FUNCTION_BLOCK ResetXYPos (* Composite Function Block Type *)
  (* Standard: 61499-2 *)
  (* Version 1.0, 2020-02-03, Mario *)
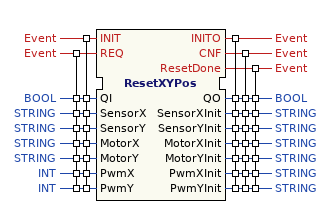
  EVENT_INPUT
    INIT WITH QI, SensorX, SensorY, MotorX, MotorY, PwmX, PwmY; (* Initialization Request *)
    REQ WITH QI, SensorX, SensorY, MotorX, MotorY, PwmX, PwmY; (* Normal Execution Request *)
  END_EVENT
  EVENT_OUTPUT
    INITO WITH QO, SensorXInit, SensorYInit, MotorXInit, MotorYInit, PwmXInit, PwmYInit; (* Initialization Confirm *)
    CNF WITH QO, SensorXInit, SensorYInit, MotorXInit, MotorYInit, PwmXInit, PwmYInit; (* Execution Confirmation *)
    ResetDone WITH QO, SensorXInit, SensorYInit, MotorXInit, MotorYInit, PwmXInit, PwmYInit;
  END_EVENT
  VAR_INPUT
    QI : BOOL; (* Input event qualifier *)
    SensorX : STRING; (* Sensor port to reset X axis *)
    SensorY : STRING; (* Sensor port to reset Y axis *)
    MotorX : STRING; (* Motor port to reset X axis *)
    MotorY : STRING; (* Motor port to reset Y axis *)
    PwmX : INT; (* Set how fast X axis should move *)
    PwmY : INT; (* Set how fast Y axis should move *)
  END_VAR
  VAR_OUTPUT
    QO : BOOL; (* Output event qualifier *)
    SensorXInit : STRING; (* Useful in debugging to check if sensorX was initialized correctly *)
    SensorYInit : STRING; (* Useful in debugging to check if sensorY was initialized correctly *)
    MotorXInit : STRING; (* Useful in debugging to check if motorX was initialized correctly *)
    MotorYInit : STRING; (* Useful in debugging to check if motorY was initialized correctly *)
    PwmXInit : STRING; (* Useful in debugging to check if motorX pwm was initialized correctly *)
    PwmYInit : STRING; (* Useful in debugging to check if motorY pwm was initialized correctly *)
  END_VAR
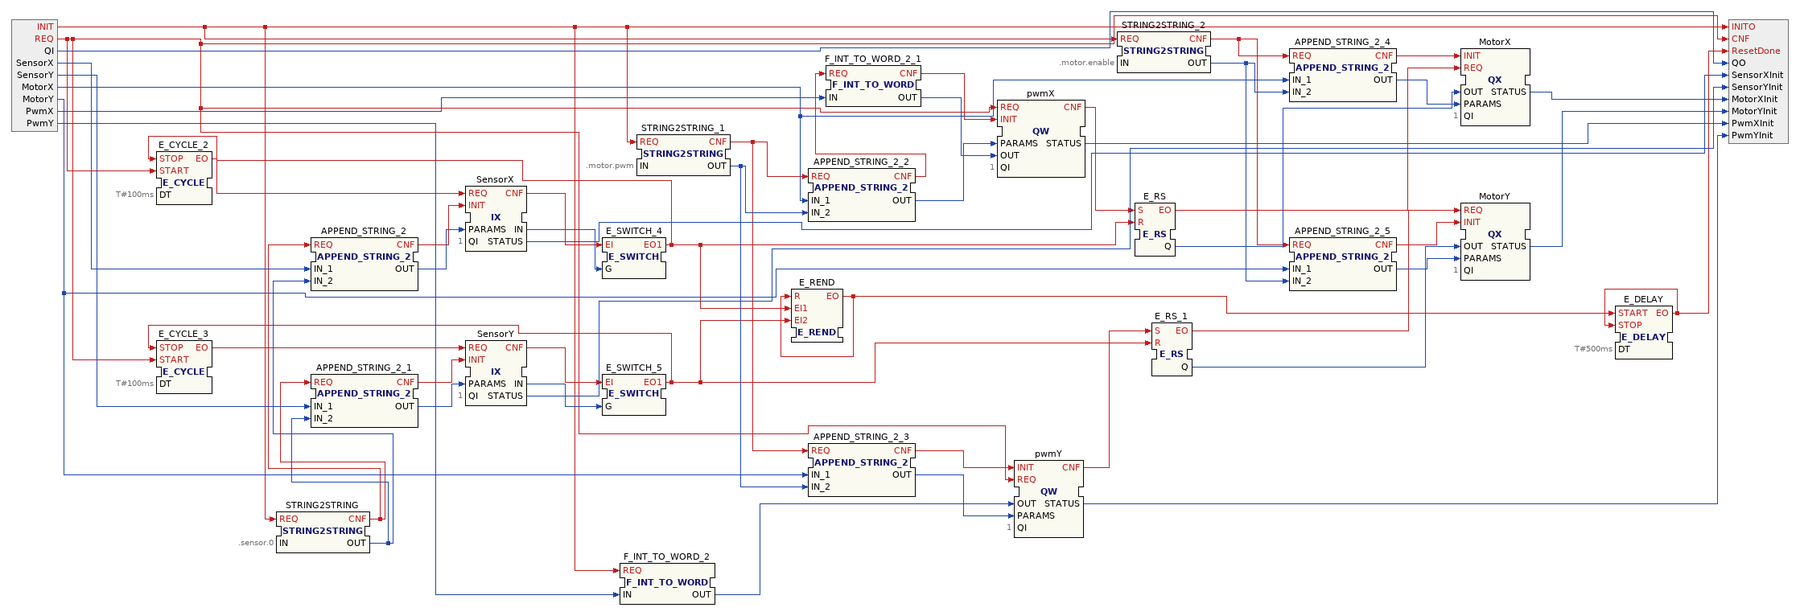
  FBS
    MotorY : QX(QI := 1);
    E_CYCLE_2 : E_CYCLE(DT := T#100ms);
    E_RS : E_RS;
    SensorY : IX(QI := 1);
    E_SWITCH_4 : E_SWITCH;
    SensorX : IX(QI := 1);
    E_REND : E_REND;
    pwmY : QW(QI := 1);
    E_CYCLE_3 : E_CYCLE(DT := T#100ms);
    E_SWITCH_5 : E_SWITCH;
    E_RS_1 : E_RS;
    F_INT_TO_WORD_2 : F_INT_TO_WORD;
    MotorX : QX(QI := 1);
    pwmX : QW(QI := 1);
    APPEND_STRING_2 : APPEND_STRING_2;
    APPEND_STRING_2_1 : APPEND_STRING_2;
    APPEND_STRING_2_2 : APPEND_STRING_2;
    APPEND_STRING_2_3 : APPEND_STRING_2;
    APPEND_STRING_2_4 : APPEND_STRING_2;
    APPEND_STRING_2_5 : APPEND_STRING_2;
    STRING2STRING : STRING2STRING(IN := .sensor.0);
    STRING2STRING_1 : STRING2STRING(IN := .motor.pwm);
    STRING2STRING_2 : STRING2STRING(IN := .motor.enable);
    F_INT_TO_WORD_2_1 : F_INT_TO_WORD;
    E_DELAY : E_DELAY(DT := T#500ms);
  END_FBS
  EVENT_CONNECTIONS
    INIT TO INITO;
    pwmX.CNF TO E_RS.S;
    pwmY.CNF TO E_RS_1.S;
    E_SWITCH_4.EO1 TO E_CYCLE_2.STOP;
    E_REND.EO TO E_REND.R;
    E_SWITCH_5.EO1 TO E_CYCLE_3.STOP;
    E_SWITCH_4.EO1 TO E_REND.EI1;
    E_SWITCH_4.EO1 TO E_RS.R;
    E_CYCLE_3.EO TO SensorY.REQ;
    SensorY.CNF TO E_SWITCH_5.EI;
    E_SWITCH_5.EO1 TO E_REND.EI2;
    E_CYCLE_2.EO TO SensorX.REQ;
    E_SWITCH_5.EO1 TO E_RS_1.R;
    SensorX.CNF TO E_SWITCH_4.EI;
    E_RS_1.EO TO MotorY.REQ;
    STRING2STRING.CNF TO APPEND_STRING_2_1.REQ;
    STRING2STRING.CNF TO APPEND_STRING_2.REQ;
    APPEND_STRING_2.CNF TO SensorX.INIT;
    APPEND_STRING_2_1.CNF TO SensorY.INIT;
    STRING2STRING_1.CNF TO APPEND_STRING_2_2.REQ;
    STRING2STRING_1.CNF TO APPEND_STRING_2_3.REQ;
    APPEND_STRING_2_3.CNF TO pwmY.INIT;
    INIT TO STRING2STRING.REQ;
    INIT TO STRING2STRING_1.REQ;
    INIT TO STRING2STRING_2.REQ;
    STRING2STRING_2.CNF TO APPEND_STRING_2_4.REQ;
    STRING2STRING_2.CNF TO APPEND_STRING_2_5.REQ;
    APPEND_STRING_2_4.CNF TO MotorX.INIT;
    APPEND_STRING_2_5.CNF TO MotorY.INIT;
    REQ TO E_CYCLE_2.START;
    REQ TO E_CYCLE_3.START;
    REQ TO pwmX.REQ;
    REQ TO pwmY.REQ;
    REQ TO CNF;
    INIT TO F_INT_TO_WORD_2.REQ;
    APPEND_STRING_2_2.CNF TO F_INT_TO_WORD_2_1.REQ;
    F_INT_TO_WORD_2_1.CNF TO pwmX.INIT;
    E_RS.EO TO MotorX.REQ;
    E_REND.EO TO E_DELAY.START;
    E_DELAY.EO TO E_DELAY.STOP;
    E_DELAY.EO TO ResetDone;
  END_CONNECTIONS
  DATA_CONNECTIONS
    F_INT_TO_WORD_2.OUT TO pwmY.OUT;
    E_RS_1.Q TO MotorY.OUT;
    E_RS.Q TO MotorX.OUT;
    SensorY.IN TO E_SWITCH_5.G;
    SensorX.IN TO E_SWITCH_4.G;
    SensorX TO APPEND_STRING_2.IN_1;
    SensorY TO APPEND_STRING_2_1.IN_1;
    MotorX TO APPEND_STRING_2_2.IN_1;
    MotorY TO APPEND_STRING_2_3.IN_1;
    MotorX TO APPEND_STRING_2_4.IN_1;
    MotorY TO APPEND_STRING_2_5.IN_1;
    STRING2STRING.OUT TO APPEND_STRING_2_1.IN_2;
    STRING2STRING.OUT TO APPEND_STRING_2.IN_2;
    APPEND_STRING_2.OUT TO SensorX.PARAMS;
    APPEND_STRING_2_1.OUT TO SensorY.PARAMS;
    STRING2STRING_1.OUT TO APPEND_STRING_2_2.IN_2;
    STRING2STRING_1.OUT TO APPEND_STRING_2_3.IN_2;
    APPEND_STRING_2_2.OUT TO pwmX.PARAMS;
    APPEND_STRING_2_3.OUT TO pwmY.PARAMS;
    STRING2STRING_2.OUT TO APPEND_STRING_2_4.IN_2;
    STRING2STRING_2.OUT TO APPEND_STRING_2_5.IN_2;
    APPEND_STRING_2_4.OUT TO MotorX.PARAMS;
    APPEND_STRING_2_5.OUT TO MotorY.PARAMS;
    QI TO QO;
    PwmY TO F_INT_TO_WORD_2.IN;
    PwmX TO F_INT_TO_WORD_2_1.IN;
    F_INT_TO_WORD_2_1.OUT TO pwmX.OUT;
    MotorX.STATUS TO MotorXInit;
    MotorY.STATUS TO MotorYInit;
    pwmY.STATUS TO PwmYInit;
    pwmX.STATUS TO PwmXInit;
    SensorX.STATUS TO SensorXInit;
    SensorY.STATUS TO SensorYInit;
  END_CONNECTIONS
END_FUNCTION_BLOCK
